// TIA Portal V20 export
DATA_BLOCK "BK02"   // DB304
// stored: MemoryReserve 100
   VAR
      "X10-1.SUCTION PAD TOP DOWN" : Bool := TRUE;
      "X11-1.SUCTION PAD BTM DOWN" : Bool := TRUE;
      "X12-1.CUTTER DOWN" : Bool := TRUE;
      "X13-1.TAPE TOP DOWN" : Bool := FALSE;
      "X14-1.TAPE BTM DOWN" : Bool := TRUE;
      "X15-1.SPLICE HEAD ROTATE TOP BACKWARD" : Bool := TRUE;
      "X16-1.SPLICE HEAD ROTATE BTM BACKWARD" : Bool := TRUE;
      "X17-1.SPARE" : Bool := FALSE;
      "X10-2.SUCTION PAD TOP UP" : Bool := FALSE;
      "X11-2.SUCTION PAD BTM UP" : Bool := FALSE;
      "X12-2.CUTTER UP" : Bool := FALSE;
      "X13-2.TAPE TOP UP" : Bool := TRUE;
      "X14-2.TAPE BTM UP" : Bool := FALSE;
      "X15-2.SPLICE HEAD ROTATE TOP FORWARD" : Bool := FALSE;
      "X16-2.SPLICE HEAD ROTATE BTM FORWARD" : Bool := FALSE;
      "X17-2.SPARE" : Bool := FALSE;
   END_VAR
BEGIN
END_DATA_BLOCK
